# EPICS autosave request: OxInstCryojet/cryojetITC503S_settings.req
$(P)$(Q):ACTIVITY:SET
$(P)$(Q):CTRL:SET
$(P)$(Q):D:SET
$(P)$(Q):DISABLE
$(P)$(Q):GFLOW:SET
$(P)$(Q):I:SET
$(P)$(Q):MANV:SET
$(P)$(Q):MAXV:SET
$(P)$(Q):P:SET
$(P)$(Q):TTEMP:SET
